{attribute 'hide_all_locals'}
FUNCTION_BLOCK FB_MotorManualCtrl

VAR_INPUT
	bForward	: BOOL;
	bBackward	: BOOL;
	bStop		: BOOL;
	Hold		: BOOL;	//Add for holding the cylinder
	Motor		: REFERENCE TO  FB_Motor; 
END_VAR
VAR_OUTPUT
END_VAR
VAR
	ForWardrTrig	:R_TRIG;
	ForWardfTrig	:F_TRIG;
	
	BackWardrTrig	:R_TRIG;
	BackWardfTrig	:F_TRIG;
	
	
	
END_VAR

IF NOT Hold THEN
	ForWardrTrig(CLK:=bForward);
	ForWardfTrig(CLK:=bForward);
	
	BackWardrTrig(CLK:=bBackward);
	BackWardfTrig(CLK:=bBackward);
END_IF

IF ForWardrTrig.Q AND NOT bBackward AND NOT bStop THEN
	Motor.M_MoveForward();	
END_IF

IF BackWardrTrig.q AND NOT bForward AND NOT bStop THEN
	Motor.M_MoveBackward();
END_IF

IF bStop OR ForWardfTrig.Q OR BackWardfTrig.Q THEN
	Motor.M_MotorStop();
END_IF

END_FUNCTION_BLOCK

(* stored: Version 1.1.0.1, ProductVersion 3.1.4024.13
   POU FB_MotorManualCtrl: Id {3c4ea09c-99de-4c83-9912-c829cfd5027c}, SpecialFunc None *)
